{attribute 'pack_mode' := '2'}
TYPE ST_XPU_STATE :
STRUCT
  Init            : E_XPU_INIT;
  State           : E_XPU_STATE;
  Check           : E_XPU_CHECK;  // cyclic check result
  DcLink          : BIT;          // power all motor modules is ON
END_STRUCT
END_TYPE

(* stored: Version 1.1.0.1, ProductVersion 3.1.4026.18
   DUT ST_XPU_STATE: Id {6d37a76d-12be-404c-85a0-5e1485f3c2bb} *)
